// TIA Portal V19 export
TYPE "SinamicsCU_Alarms"
// stored: Access Published
   STRUCT
      CUFault : Bool;   // Fault from CU telegram
      CommunicationFault : Bool;   // Communication fault
   END_STRUCT;
END_TYPE
